PROGRAM PRG_AL1L0_REF
VAR
    {attribute 'pytmc' := 'pv: AL1L0:REF'}
    {attribute 'TcLinkTo' := '.fbLaser.iLaserINT := TIIB[AL1L0-EL4004-E4]^AO Outputs Channel 3^Analog output;
                              .fbLaser.iShutdownINT := TIIB[AL1L0-EL4004-E4]^AO Outputs Channel 2^Analog output'}
    fbAL1L0: FB_REF;

    fbStateSetup: FB_StateSetupHelper;
    stDefault: ST_PositionState := (
        fVelocity := 1,
        bMoveOk := TRUE,
        bValid := TRUE
    );
END_VAR

//Device doesn't have end of travel limits switches
MAIN.M58.bLimitBackwardEnable := TRUE;
MAIN.M58.bLimitForwardEnable := TRUE;


fbStateSetup(stPositionState:=stDefault, bSetDefault:=TRUE);
fbStateSetup(stPositionState:=fbAL1L0.stOut, fPosition:=0, sPmpsState:='AL1L0:REF-OUT');
fbStateSetup(stPositionState:=fbAL1L0.stIn, fPosition:=-43.38, fDelta:=2, sPmpsState:='AL1L0:REF-IN');

fbAL1L0(
    fbFFHWO := GVL.fbFastFaultOutput1d,
    fbArbiter := GVL.fbArbiter,
    stYStage := MAIN.M58,
    sDeviceName := 'AL1L0:REF',
    sTransitionKey := 'AL1L0:REF-TRANSITION',
    bEnableMotion := TRUE,
    bEnableBeamParams := TRUE,
    bEnablePositionLimits := TRUE,
);
// Needed to prevent gravity from pulling the stage down since there is no brake
MAIN.M58.nEnableMode := ENUM_StageEnableMode.ALWAYS;

END_PROGRAM

(* stored: Version 1.1.0.1
   POU PRG_AL1L0_REF: Id {0d63d84a-166a-0041-1034-84e836973389}, SpecialFunc None *)
